// TwinCAT 3 PLC project example
// ProgramVersion: 3.1.4026.12
// libraries:
//   Tc2_Standard, * (Beckhoff Automation GmbH)
//   Tc2_System, * (Beckhoff Automation GmbH)
// project tree:
//   / PlcTask.TcTTO
//   POUs/ MAIN.TcPOU
// (motion and I/O tree: see PLC project plcudpserver)
// real-time tasks:
//   TASK PlcTask: cycle T#1ms, priority 23, ADS port 350
//   TASK PlcTask1: cycle T#10ms, priority 20, ADS port 351
// variable links:
//   example/example Instance <-> Device 1 (EtherCAT)/Term 1 (EK1200)/Term 2 (EL6695)
//     PlcTask Inputs/MAIN.testBoolFromROS <-> IO Inputs/BoolFromROS
//     PlcTask Inputs/MAIN.testInt32FromROS <-> IO Inputs/int32FromROS
//     PlcTask Outputs/MAIN.testBoolToROS <-> IO Outputs/BoolToROS
//     PlcTask Outputs/MAIN.testInt32ToROS <-> IO Outputs/int32ToROS

CONFIGURATION example
    RESOURCE PLC ON TwinCAT3
        TASK PlcTask(INTERVAL := T#10ms, PRIORITY := 20);
        PROGRAM MAIN WITH PlcTask : MAIN;
    END_RESOURCE
END_CONFIGURATION

// ---- POUs/MAIN.TcPOU
PROGRAM MAIN
VAR
	testInt32ToROS AT %Q* :DINT :=0 ;
	testBoolToROS AT %Q*:BOOL :=TRUE;
	testInt32FromROS AT %I* :DINT :=0;
	testBoolFromROS AT %I*:BOOL:=FALSE;
END_VAR

testInt32ToROS := testInt32ToROS+1;

END_PROGRAM
